// SIMATIC S7-200 project (STEP 7-Micro/WIN), CPU 224XP CN REL 02.01

SYMBOL_TABLE USER1
wOpenRateFb      VW0      // 开度反馈
wOpenRateRf      VW2      // 开度设置
dActionCount     VD4      // 动作计数
aiOpenRateFb     AIW2     // 开度反馈输入
aqOpenRateRf     AQW0     // 开度设置输出
END_SYMBOL_TABLE

ORGANIZATION_BLOCK MAIN:OB1
TITLE=PROGRAM COMMENTS
BEGIN
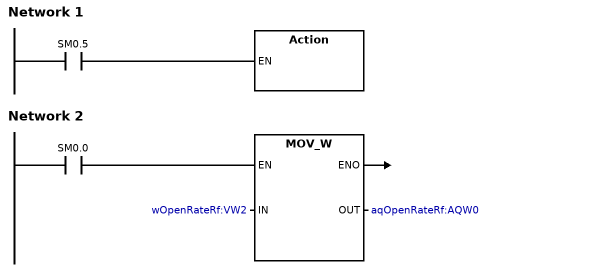
Network 1
LD     SM0.5
CALL   Action:SBR0
Network 2
LD     SM0.0
MOVW   wOpenRateRf:VW2, aqOpenRateRf:AQW0
END_ORGANIZATION_BLOCK

SUBROUTINE_BLOCK Action:SBR0
TITLE=SUBROUTINE COMMENTS
BEGIN
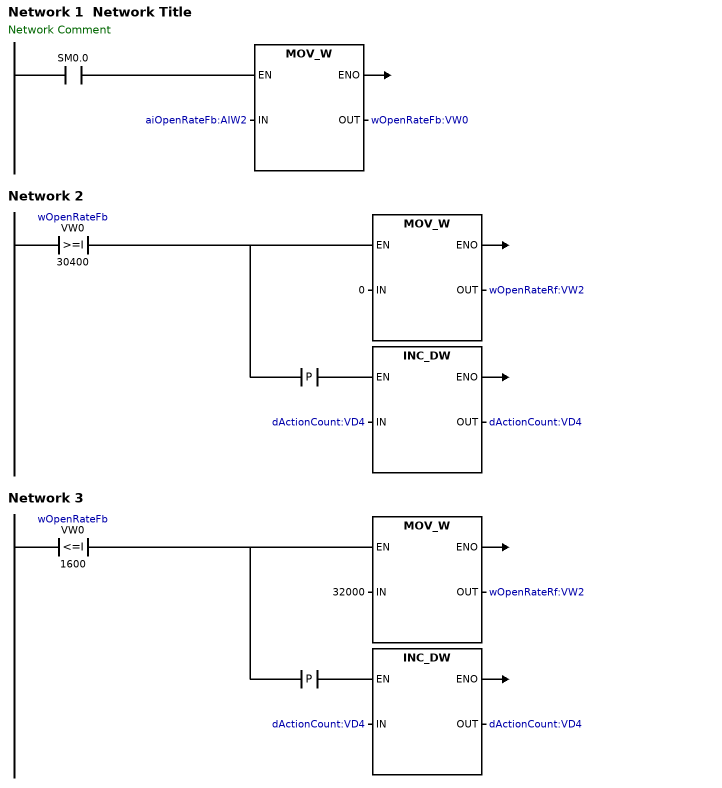
Network 1 // Network Title
// Network Comment
LD     SM0.0
MOVW   aiOpenRateFb:AIW2, wOpenRateFb:VW0
Network 2
// (network saved uncompiled; LAD cells follow)
// row 0: c0 -|>=I|- wOpenRateFb:VW0, 30400  c1 -- v  c2 --  c3 [MOV_W EN:=power@row0, IN:=0, ENO=>power, OUT=>wOpenRateRf:VW2]  c4 ->
// row 1: c1 ^v  c3 [box]
// row 2: c1 ^  c2 -|P|-  c3 [INC_DW EN:=power@row2, IN:=dActionCount:VD4, ENO=>power, OUT=>dActionCount:VD4]  c4 ->
// row 3: c3 [box]
Network 3
// (network saved uncompiled; LAD cells follow)
// row 0: c0 -|<=I|- wOpenRateFb:VW0, 1600  c1 -- v  c2 --  c3 [MOV_W EN:=power@row0, IN:=32000, ENO=>power, OUT=>wOpenRateRf:VW2]  c4 ->
// row 1: c1 ^v  c3 [box]
// row 2: c1 ^  c2 -|P|-  c3 [INC_DW EN:=power@row2, IN:=dActionCount:VD4, ENO=>power, OUT=>dActionCount:VD4]  c4 ->
// row 3: c3 [box]
END_SUBROUTINE_BLOCK
